FUNCTION_BLOCK RunAxis EXTENDS CommonBase
VAR_OUTPUT
	PositionFeedback : LREAL;
	//PositionCommand : LREAL;
END_VAR
VAR	
	Axis : AXIS_REF;
	 
	nCounter : int :=0;
	fbMoveAbs : ARRAY[1..3] OF MC_MoveAbsolute; //preset n buffers available
	fbMoveHome : MC_Home;
	fbPower : MC_Power;
	fbReset: MC_Reset;
	fbSetPosition: MC_SetPosition;
	
	//Status reading
	fbReadActualVelocity: MC_ReadParameter;
	fbReadActualPosition : MC_ReadActualPosition;
	fbReadCommandPosition : MC_ReadParameter;
	fbReadStatus : MC_ReadStatus;
	//Parameter writing
	fbWriteLimitPositive : MC_WriteParameter;
	fbWriteLimitNegtive : MC_WriteParameter;
	
	timerFbReset : TON;
	//bMonitoring : bool;
END_VAR
VAR PERSISTENT
	ptpCommands : ARRAY[1..12] OF ParameterSet; //collect command blocks relative to this axis here
END_VAR
VAR CONSTANT
	typeCode : eCategrories := eCategrories.SELECTION_AXIS;
END_VAR

//----------------------------SW Limit
fbWriteLimitPositive(
	Axis:= Axis, 
	Execute:= , 
	ParameterNumber:= SWLimitPos, 
	Value:= , 
	Done=> , 
	Busy=> , 
	Error=> , 
	ErrorID=> );
IF fbWriteLimitPositive.Execute AND (fbWriteLimitPositive.Done OR fbWriteLimitPositive.Error) THEN
	fbWriteLimitPositive.Execute := FALSE; //auto reset
END_IF
fbWriteLimitNegtive(
	Axis:= Axis, 
	Execute:= , 
	ParameterNumber:= SWLimitNeg, 
	Value:= , 
	Done=> , 
	Busy=> , 
	Error=> , 
	ErrorID=> );
IF fbWriteLimitNegtive.Execute AND (fbWriteLimitNegtive.Done OR fbWriteLimitNegtive.Error) THEN
	fbWriteLimitNegtive.Execute := FALSE;
END_IF
//----------------------------

fbReadCommandPosition(
	Axis:= Axis, 
	Enable:= TRUE, 
	ParameterNumber:= CommandedPosition, 
	ReadMode:= READMODE_CYCLIC, 
	Valid=> , 
	Busy=> , 
	Error=> , 
	ErrorID=> , 
	Value=> );


fbSetPosition(
	Axis:= Axis, 
	Execute:= , 
	Position:= , 
	Mode:= , 
	Options:= , 
	Done=> , 
	Busy=> , 
	Error=> , 
	ErrorID=> );

//default mode
fbPower(
	Axis:= Axis, 
	Enable:= , 
	Enable_Positive:= , 
	Enable_Negative:= , 
	Override:= , 
	BufferMode:= , 
	Options:= , 
	Status=> , 
	Busy=> , 
	Active=> , 
	Error=> , 
	ErrorID=> );
	
fbReset(
	Axis:= Axis, 
	Execute:= , 
	Done=> , 
	Busy=> , 
	Error=> , 
	ErrorID=> );

// Reset alarm clear after 100ms
timerFbReset(IN:= fbReset.Execute, PT:= T#100MS, Q=> , ET=> );	
IF timerFbReset.Q THEN
	fbReset.Execute := FALSE;
END_IF
	
//Status reading and update
fbReadActualVelocity(
	Axis:= Axis, 
	Enable:= TRUE, 
	ParameterNumber:= ActualVelocity, 
	ReadMode:= READMODE_CYCLIC, 
	Valid=> , 
	Busy=> , 
	Error=> , 
	ErrorID=> , 
	Value=> );

fbReadActualPosition(
	Axis:= axis, 
	Enable:= TRUE, 
	Valid=> , 
	Busy=> , 
	Error=> , 
	ErrorID=> , 
	Position=> PositionFeedback);

fbReadStatus(
	Axis:= axis, 
	Enable:= TRUE, 
	Valid=> , 
	Busy=> , 
	Error=> , 
	ErrorID=> , 
	ErrorStop=> , 
	Disabled=> , 
	Stopping=> , 
	StandStill=> , 
	DiscreteMotion=> , 
	ContinuousMotion=> , 
	SynchronizedMotion=> , 
	Homing=> , 
	ConstantVelocity=> , 
	Accelerating=> , 
	Decelerating=> , 
	Status=> );
	
IF NOT fbPower.Enable THEN
	RETURN; //do not execute following commands
END_IF
	//execute founction blocks once powered
	//possible to configure how many buffer used
	FOR nCounter:=1 TO 3 BY 1 DO
	fbMoveAbs[nCounter](
		Axis:= Axis, 
		Execute:= , 
		Position:= , 
		Velocity:= , 
		Acceleration:= , 
		Deceleration:= , 
		Jerk:= , 
		BufferMode:= MC_BlendingPrevious, 
		Options:= , 
		Done=> , 
		Busy=> , 
		Active=> , 
		CommandAborted=> , 
		Error=> , 
		ErrorID=> );
	END_FOR
	
		
	fbMoveHome(
		Axis:= Axis, 
		Execute:= , 
		Position:= , 
		HomingMode:= , 
		BufferMode:= , 
		Options:= , 
		bCalibrationCam:= , 
		Done=> , 
		Busy=> , 
		Active=> , 
		CommandAborted=> , 
		Error=> , 
		ErrorID=> );

METHOD ConfigureRead : CellDataBlock
VAR_INPUT
	mode : eModes;
END_VAR
END_METHOD

METHOD ConfigureWrite : BOOL
VAR_INPUT
	input : CellDataBlock;
	mode : eModes;
END_VAR
VAR
	temp : ParameterSet; 
END_VAR
//command block write-in
CASE mode OF
	eModes.MODE_EXE_AXIS:
		//software limit
		fbWriteLimitPositive.Value := TO_REAL(input.axis.limitPlus) * 0.001;
		fbWriteLimitPositive.Execute := TRUE;
		
		fbWriteLimitNegtive.Value := TO_REAL(input.axis.limitMinus) * 0.001;
		fbWriteLimitNegtive.Execute := TRUE;
		
	eModes.MODE_EXE_COMMAND_BLOCK:
		temp := CellDataBlock2Parameter(input:= input);
		ptpCommands[input.command.base.subIndex+1] := temp; //write-in
		
END_CASE

ConfigureWrite := TRUE; //return
END_METHOD

METHOD Control : BOOL
VAR_INPUT
	input : CellDataBlock;
	mode : eModes;
END_VAR
VAR
	temp : ParameterSet;
END_VAR
//manual control servo on/servo alarm reset

//different route
CASE mode OF
	eModes.MODE_EXE_AXIS:
		IF input.axis.operationOperation.0 THEN
			//bit0ServoOn
			fbPower.Enable := NOT fbPower.Enable;
			fbPower.Enable_Positive := fbPower.Enable;
			fbPower.Enable_Negative := fbPower.Enable;
		ELSIF input.axis.operationOperation.15 THEN
			fbReset.Execute := TRUE;	
		END_IF
		Control := TRUE;
	eModes.MODE_EXE_COMMAND_BLOCK:
		temp := CellDataBlock2Parameter(input:= input);
		Control := ExecuteParameter(ptBlock:= ADR(temp));
END_CASE
END_METHOD

METHOD ErrorClear : BOOL
VAR_INPUT
	input : eErrorClearWays;
END_VAR
CASE input OF
	eErrorClearWays.RESET:
		fbReset.Execute := true;
END_CASE
END_METHOD

METHOD ErrorDetect : UDINT
VAR_INPUT
END_VAR
ErrorDetect := fbReadStatus.ErrorID;
END_METHOD

METHOD ExecuteParameter : BOOL
VAR_INPUT
	ptBlock : POINTER TO ParameterSet;
	//execute : BOOL; //used to do mutex
END_VAR
//
ExecuteParameter:=ExecuteParameterBuffer(ptBlock:= ptBlock, bufferIndex:= 1);
END_METHOD

METHOD ExecuteParameterBuffer : BOOL
VAR_INPUT
	ptBlock : POINTER TO ParameterSet;
	//execute : BOOL; //used to do mutex
	bufferIndex: INT :=1;
END_VAR
VAR
	//MC block routing
	ptMcExecute : POINTER TO BOOL;
	ptMcDone : POINTER TO BOOL;
	ptMcBusy : POINTER TO BOOL;
	ptMcError : POINTER TO BOOL;
	ptMcCommandAbort : POINTER TO BOOL;

END_VAR
//1. Do parameter translating
//2. Do command routing
//3. Control execute flow

//command routing
CASE ptBlock^.command OF
eCommandTypes.POSITION:	
	//Position command
	ptMcExecute:=ADR(fbMoveAbs[bufferIndex].Execute);
	ptMcDone:=ADR(fbMoveAbs[bufferIndex].Done);
	ptMcBusy:=ADR(fbMoveAbs[bufferIndex].Busy);
	ptMcError:=ADR(fbMoveAbs[bufferIndex].Error);
	ptMcCommandAbort := ADR(fbMoveAbs[bufferIndex].CommandAborted);
	//set once
	IF NOT fbMoveAbs[bufferIndex].Busy AND NOT ptMcExecute^ THEN
		//parameter writing
		fbMoveAbs[bufferIndex].Velocity := ptBlock^.parameter.position.Velocity;
		fbMoveAbs[bufferIndex].Acceleration:= ptBlock^.parameter.position.Acceleration;
		fbMoveAbs[bufferIndex].Deceleration:= ptBlock^.parameter.position.Deceleration;
		
		CASE ptBlock^.parameter.position.PositionType OF
			ePositionType.POSITION_ABS:
				fbMoveAbs[bufferIndex].Position := ptBlock^.parameter.position.Position;
			ePositionType.POSITION_REL:
				fbMoveAbs[bufferIndex].Position := PositionCommand + ptBlock^.parameter.position.Position; 
		END_CASE
		
	END_IF
	
	IF bufferIndex>=2 THEN
		fbMoveAbs[bufferIndex].BufferMode := MC_BlendingPrevious;
	END_IF
//torque limit
;
eCommandTypes.ZRET:
	//Home command
	ptMcExecute:=ADR(fbMoveHome.Execute);
	ptMcDone:=ADR(fbMoveHome.Done);
	ptMcBusy:=ADR(fbMoveHome.Busy);
	ptMcError:=ADR(fbMoveHome.Error);
	ptMcCommandAbort := ADR(fbMoveHome.CommandAborted);
	
	IF NOT fbMoveHome.Busy THEN
		//parameter writing
		fbMoveHome.Position := ptBlock^.parameter.home.Position;
		fbMoveHome.HomingMode := ptBlock^.parameter.home.Mode;
	END_IF
;
eCommandTypes.SET_POSITION:
	ptMcExecute:=ADR(fbSetPosition.Execute);
	ptMcDone:=ADR(fbSetPosition.Done);
	ptMcBusy:=ADR(fbSetPosition.Busy);
	ptMcError:=ADR(fbSetPosition.Error);
	ptMcCommandAbort := ADR(fbSetPosition.Done);// fake
	
	IF NOT fbSetPosition.Busy THEN
		//parameter writing
		fbSetPosition.Position := ptBlock^.parameter.position.Position;
	END_IF
	
ELSE
	return;
END_CASE

//auto stop execute when error , would do raising edge again when error eliminated
ptMcExecute^ := NOT ptMcError^ AND NOT ptMcDone^ AND NOT ptMcCommandAbort^;

//power on if going to execute
IF ptMcExecute^ AND fbPower.Enable=FALSE THEN
	fbPower.Enable := TRUE;
	fbPower.Enable_Positive := TRUE;
	fbPower.Enable_Negative := TRUE;
END_IF

//done := ptMcDone^;
ExecuteParameterBuffer:=ptMcDone^; //return value
END_METHOD

METHOD ExecuteParameterBufferIndex : BOOL
VAR_INPUT
	indexCommand : INT ;
	indexBuffer : INT;
END_VAR
//wrapper function
ExecuteParameterBufferIndex := ExecuteParameterBuffer(ptBlock:= ADR(ptpCommands[indexCommand]), bufferIndex:= indexBuffer);
END_METHOD

METHOD ExecuteParameterIndex : BOOL
VAR_INPUT
	indexCommand : int;
END_VAR
//wrpper function 
ExecuteParameterIndex:=ExecuteParameter(ptBlock:= adr(ptpCommands[indexCommand]));
END_METHOD

METHOD FB_init : BOOL
VAR_INPUT
	bInitRetains : BOOL; // if TRUE, the retain variables are initialized (warm start / cold start)
	bInCopyCode : BOOL;  // if TRUE, the instance afterwards gets moved into the copy code (online change)
END_VAR
VAR
	nCounter : int ;
END_VAR
END_METHOD

METHOD Monitor : CellDataBlock
VAR_INPUT
END_VAR
Monitor.axis.operationMonitor.0 := fbPower.Enable;
Monitor.axis.operationMonitor.15 := fbReset.Execute;

Monitor.axis.runStatus.1 := fbReadStatus.StandStill;
Monitor.axis.runStatus.3 := not fbReadStatus.Error;

Monitor.axis.alarm := fbReadStatus.ErrorID;

Monitor.axis.posCommand := TO_DINT(fbReadCommandPosition.Value * 1000);
Monitor.axis.posFeedback := TO_DINT(fbReadActualPosition.Position * 1000);
Monitor.axis.speedFeedback := TO_DINT(fbReadActualVelocity.Value * 1000);
END_METHOD

PROPERTY PositionCommand : LREAL
GET
fbReadCommandPosition.Enable := TRUE;
//fbReadCommandPosition(
//	Axis:= Axis, 
//	Enable:= , 
//	ParameterNumber:= CommandedPosition, 
//	ReadMode:= READMODE_ONCE, 
//	Valid=> , 
//	Busy=> , 
//	Error=> , 
//	ErrorID=> , 
//	Value=> PositionCommand);
PositionCommand := fbReadCommandPosition.Value;
END_GET
SET
END_SET
END_PROPERTY

METHOD Stop : BOOL
VAR_INPUT
END_VAR
VAR
	nCounter : INT;
END_VAR
//stop all function blocks
FOR nCounter:=1 TO 3 BY 1 DO
	fbMoveAbs[nCounter].Execute := FALSE;
END_FOR
fbMoveHome.Execute := FALSE;
END_METHOD

METHOD TypeCode : eCategrories
VAR_INPUT
END_VAR
TypeCode := eCategrories.SELECTION_AXIS;
END_METHOD

END_FUNCTION_BLOCK

(* stored: Version 1.1.0.1, ProductVersion 3.1.4022.10
   POU RunAxis: Id {1e355049-017f-4f7f-88a6-a7040666a5c5}, SpecialFunc None
   Folder CommonBase: Id {7c375d8d-5198-4156-90d1-ff49df703551}
   Method ConfigureRead: Id {b2d706a8-b020-4343-983c-4c7a56c09ac2}
   Method ConfigureWrite: Id {cde8b8df-cc3c-4ac1-a00a-6c29224f2a1d}
   Method Control: Id {fb2d590a-2a78-44ed-97fd-631e13336dc9}
   Method ErrorClear: Id {3448d412-4c2e-4bc3-a590-f166f4dbcea7}
   Method ErrorDetect: Id {da618aca-91fe-4791-8fbe-90aff9c7dc94}
   Method ExecuteParameter: Id {71f56729-8e13-4b1e-a80c-858adc37a723}
   Method ExecuteParameterBuffer: Id {248fd65c-916e-4c41-b72b-91932f742cc7}
   Method ExecuteParameterBufferIndex: Id {e08cab37-7a1e-49ab-bbc7-cc8815b18348}
   Method ExecuteParameterIndex: Id {47d338d7-7440-407f-9fdb-d43303a84fa1}
   Method FB_init: Id {5aeba573-47c3-411b-9f3d-8af6b6892223}
   Method Monitor: Id {f14ef5b7-4fb3-4276-899b-459b8636a870}
   Property PositionCommand: Id {d90f9427-641f-46be-8de0-14848d24631d}
   Get Get: Id {19f01c9c-5d4f-4654-8572-382eb730f8d5}
   Set Set: Id {dd39da7a-143a-4c85-876d-cc4718cf70aa}
   Method Stop: Id {92c52b93-2b5b-43c1-8417-c41b77593d4d}
   Method TypeCode: Id {d7c803da-ddd0-409e-b8b9-d71f78281c2b} *)
